FUNCTION_BLOCK DigitalInput_NC EXTENDS Component IMPLEMENTS I_DigitalInput
VAR
	Input		  : REFERENCE TO BOOL;
	ForcibleInput : ForcibleBool(_Name);
END_VAR

//FB_Init is always available implicitly and it is used primarily for initialization.

//The return value is not evaluated. For a specific influence, you can also declare the

//methods explicitly and provide additional code there with the standard initialization

//code. You can evaluate the return value.
METHOD FB_Init : BOOL
VAR_INPUT
	bInitRetains : BOOL; // TRUE: the retain variables are initialized (reset warm / reset cold)
	bInCopyCode	 : BOOL; // TRUE: the instance will be copied to the copy code afterward (online change)   
	Name		 : T_MaxString;
	Input		 : REFERENCE TO BOOL;
END_VAR
THIS^.Input REF= Input;
END_METHOD

{attribute 'monitoring' := 'call'}
PROPERTY Force : E_ForceState
GET
Force := ForcibleInput.CurrentForceState;
END_GET
SET
VAR
	ForceString : T_MaxString := TO_STRING(Force);
END_VAR
ForcibleInput.SetForceState(Force);
END_SET
END_PROPERTY

{attribute 'monitoring' := 'call'}
PROPERTY IsActive : BOOL
GET
ForcibleInput.Input := NOT Input;
IsActive			:= ForcibleInput.Output;
END_GET
END_PROPERTY

END_FUNCTION_BLOCK

(* stored: Version 1.1.0.1, ProductVersion 3.1.4026.18
   POU DigitalInput_NC: Id {e6e54a28-ad82-4ad1-9614-af6f56f9a48b}, SpecialFunc None
   Method FB_Init: Id {12d0ef35-6330-4c23-843c-af1ae73a6200}
   Property Force: Id {4c5a5179-7d73-4714-b916-c3f71c22bdf3}
   Get Get: Id {81204393-ca12-454c-9ec5-676f2f4242c4}
   Set Set: Id {894c037b-d93f-4a44-ba14-bcf8f549c64e}
   Property IsActive: Id {ab42629a-4dc8-4e88-9e44-c5ac3c74d422}
   Get Get: Id {abf91698-86de-43c6-8243-4c07e739c18c} *)
